{attribute 'qualified_only'}
VAR_GLOBAL
	K1 AT %Q* :BOOL; // Vereinzelner
	K2 AT %Q* :BOOL; // Füllen
	P1 AT %Q* :BOOL; // Behälter leer
	Q1 AT %Q* :BOOL; // Förderband
END_VAR

(* stored: Version 1.1.0.1, ProductVersion 3.1.4024.5
   GVL DA: Id {efa3d63a-96e1-4204-b1e7-9f3703bd4f03} *)
